PROGRAM V0_4
VAR
	fbR_Trig : R_TRIG;
	bTrigger : BOOL;
END_VAR

(*
	Opslagvat
	
	Een opslagvat heeft twee sensoren in de zijwand die een laag en hoog niveau aanduiden. Aan de hand van een PLC programma dient er
	automatisch de klep bovenaan het vat geopend te worden als het vat leeg is. De tank wordt nu gevuld. Als de tank vol is
	sluit de klep K1 eveneens automatisch. Onderaan de tank bevindt zich een pomp P1 die met een start- en stop-drukknop in- en
	uitgeschakeld kan worden. 

	Als de tank leeg gelopen is, stopt de pomp automatisch en opent de klep K1 bovenaan. De pomp kan niet ingeschakeld worden
	zolang de tank gevuld wordt.
	
	(T = Toggle)
	L1	l2	S1	P1	K1
	0	0	x	x	1
	1	0	x	x	1
	1	1	x	x	0
	
	x	x	0	0T	x
	x	x	1	1T	x
*)

GVL.bLamp_1 := NOT GVL.bSwitch_1; // L2

GVL.bLamp_2 R= (GVL.bButton_1 AND GVL.bLamp_2) OR (NOT GVL.bSwitch_1);
GVL.bLamp_2 S= GVL.bButton_2 AND NOT GVL.bLamp_2 AND GVL.bSwitch_1;

END_PROGRAM

(* stored: Version 1.1.0.1, ProductVersion 3.1.4024.12
   POU V0_4: Id {089e5ee0-bf9c-4577-932c-a02e27c2214b}, SpecialFunc None *)
